TYPE AstarAlgorithmusVariablen :
STRUCT
END_STRUCT
END_TYPE

(* stored: Version 1.1.0.1, ProductVersion 3.1.4024.11
   DUT AstarAlgorithmusVariablen: Id {c5854c3c-7a83-4054-a8b4-ae6c4005eaed} *)
